// SIMATIC S7-200 project (STEP 7-Micro/WIN), CPU 222 CN REL 02.01

ORGANIZATION_BLOCK 主程序:OB1
TITLE=程序注释
BEGIN
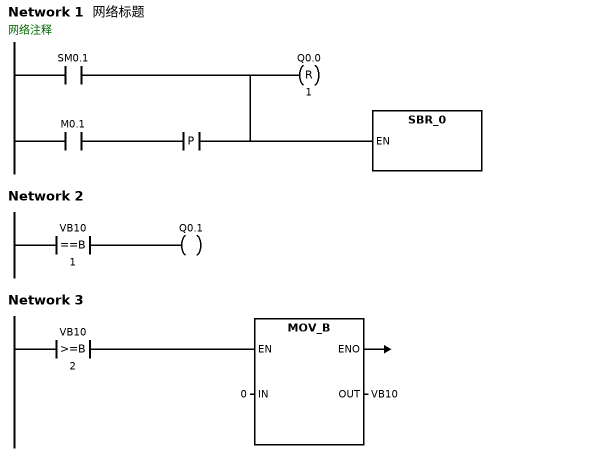
Network 1 // 网络标题
// 网络注释
LD     SM0.1
LD     M0.1
EU
OLD
R      Q0.0, 1
CALL   SBR_0:SBR0
Network 2
LDB=   VB10, 1
=      Q0.1
Network 3
LDB>=  VB10, 2
MOVB   0, VB10
END_ORGANIZATION_BLOCK

SUBROUTINE_BLOCK SBR_0:SBR0
TITLE=子程序注释
BEGIN
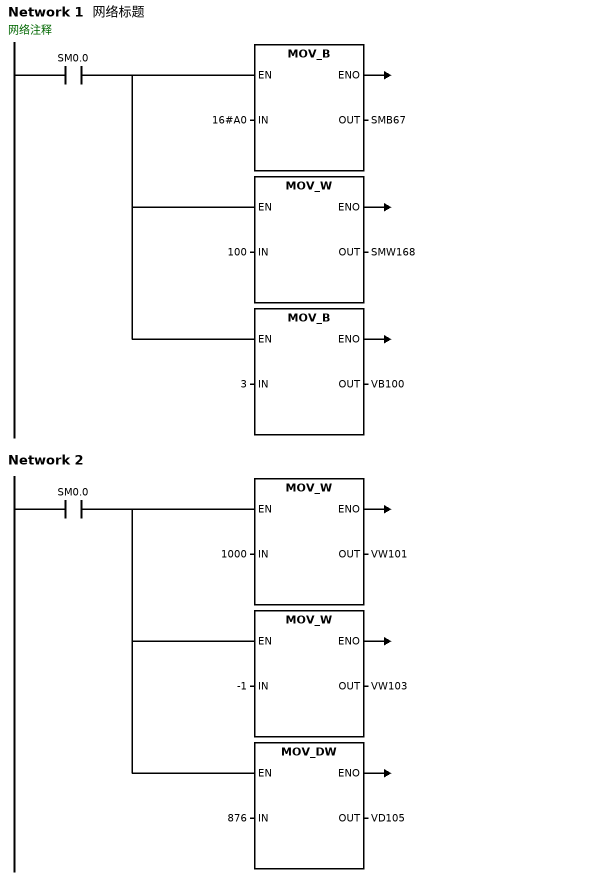
Network 1 // 网络标题
// 网络注释
LD     SM0.0
MOVB   16#A0, SMB67
MOVW   100, SMW168
MOVB   3, VB100
Network 2
LD     SM0.0
MOVW   1000, VW101
MOVW   -1, VW103
MOVD   876, VD105
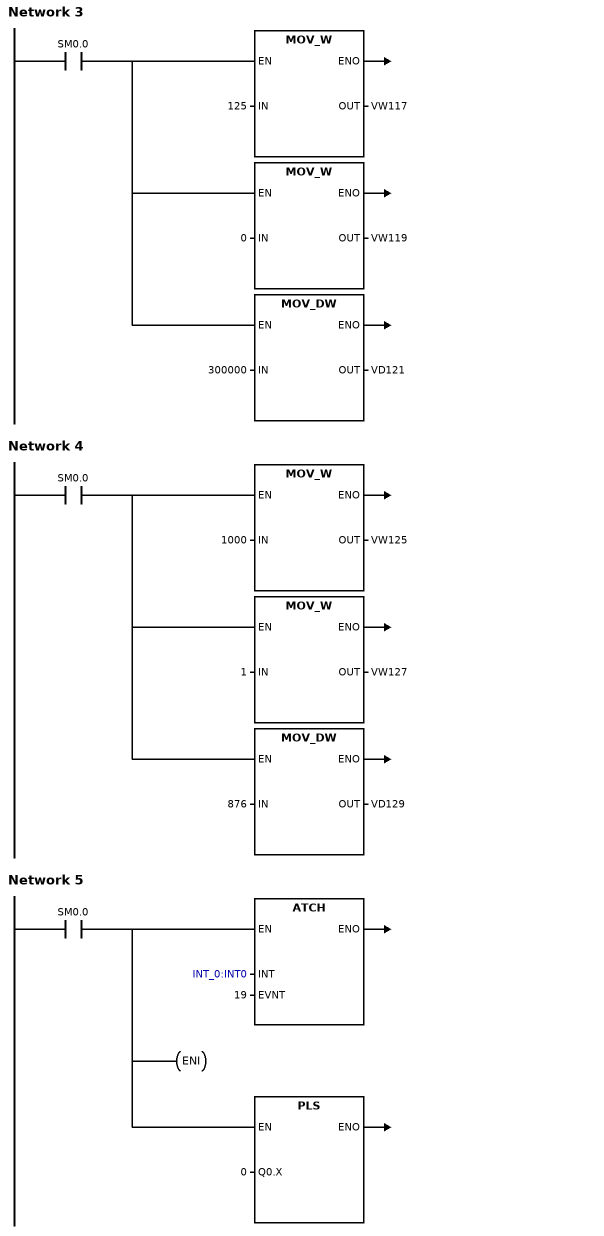
Network 3
LD     SM0.0
MOVW   125, VW117
MOVW   0, VW119
MOVD   300000, VD121
Network 4
LD     SM0.0
MOVW   1000, VW125
MOVW   1, VW127
MOVD   876, VD129
Network 5
LD     SM0.0
ATCH   INT_0:INT0, 19
ENI
PLS    0
END_SUBROUTINE_BLOCK

INTERRUPT_BLOCK INT_0:INT0
TITLE=中断程序注释
BEGIN
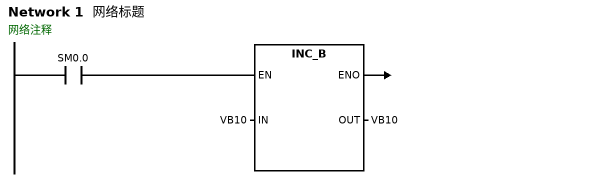
Network 1 // 网络标题
// 网络注释
LD     SM0.0
INCB   VB10
END_INTERRUPT_BLOCK
